FUNCTION_BLOCK FB_WriteParameters
VAR_INPUT
END_VAR
VAR_OUTPUT
END_VAR
VAR
END_VAR

// axis parameters offsets
// https://infosys.beckhoff.com/content/1033/tc3_ads_intro/713091211.html?id=750639462434375559

END_FUNCTION_BLOCK

(* stored: Version 1.1.0.1
   POU FB_WriteParameters: Id {354cf1fb-f624-4983-96ea-6aaa15bf364e}, SpecialFunc None *)
